PROGRAM PRG_09_PlcDiagnostic
VAR
	NetID						: 	STRING := '192.168.1.145.1.1';
	tonRecycle50ms				: 	TON;
	tonRecyclePublishMqtt		: 	TON;
	
	CpuMemoryUsage				:	ReadMemoryUsage;
	CpuUsageEx_Core2			:	TC_CPuUsageEx;
	CpuUsageEx_Core3			:	TC_CPuUsageEx;
	CpuLatencyEx_Core2			:	TC_SysLatencyEx;
	CpuLatencyEx_Core3			:	TC_SysLatencyEx;
	
	PlcDiagState				:	ARRAY [1..5] OF GenericState;
	
	{attribute 'OPC.UA.DA' := '0'}
	{attribute 'OPC.UA.DA.Access' := '1'}			// read only
	{attribute 'OPC.UA.DA.StructuredType' := '1'}
	PlcCpuMemUsageStruct		: SingleState_DataModel;
	
	{attribute 'OPC.UA.DA' := '0'}
	{attribute 'OPC.UA.DA.Access' := '1'}			// read only
	{attribute 'OPC.UA.DA.StructuredType' := '1'}
	PlcCpuCore2UsageStruct		: SingleState_DataModel;
	
	{attribute 'OPC.UA.DA' := '0'}
	{attribute 'OPC.UA.DA.Access' := '1'}			// read only
	{attribute 'OPC.UA.DA.StructuredType' := '1'}
	PlcCpuCore3UsageStruct		: SingleState_DataModel;
	
	{attribute 'OPC.UA.DA' := '0'}
	{attribute 'OPC.UA.DA.Access' := '1'}			// read only
	{attribute 'OPC.UA.DA.StructuredType' := '1'}
	PlcCpuCore2JitterStruct		: SingleState_DataModel;
	
	{attribute 'OPC.UA.DA' := '0'}
	{attribute 'OPC.UA.DA.Access' := '1'}			// read only
	{attribute 'OPC.UA.DA.StructuredType' := '1'}
	PlcCpuCore3JitterStruct		: SingleState_DataModel;

END_VAR


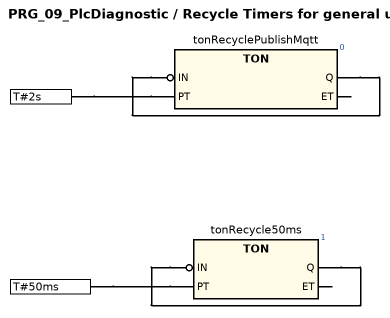
// PAGE Recycle Timers for general usage ---
tonRecyclePublishMqtt(IN := NOT tonRecyclePublishMqtt.Q, PT := T#2s); // TON
tonRecycle50ms(IN := NOT tonRecycle50ms.Q, PT := T#50ms); // TON

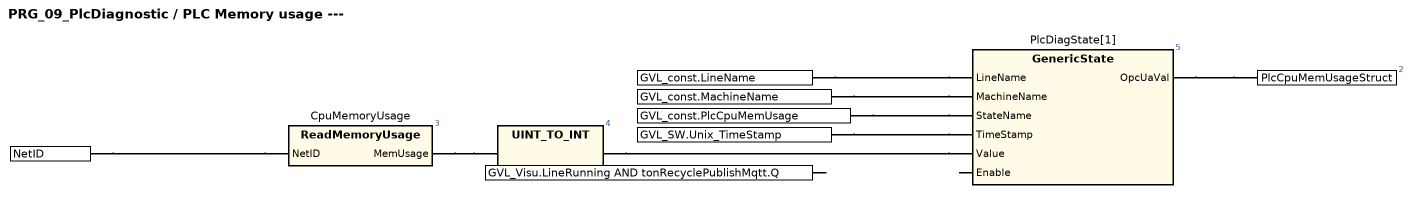
// PAGE PLC Memory usage ---
PlcCpuMemUsageStruct := PlcDiagState[1].OpcUaVal;
CpuMemoryUsage(NetID := NetID); // ReadMemoryUsage
PlcDiagState[1](
    LineName := GVL_const.LineName,
    MachineName := GVL_const.MachineName,
    StateName := GVL_const.PlcCpuMemUsage,
    TimeStamp := GVL_SW.Unix_TimeStamp,
    Value := UINT_TO_INT(CpuMemoryUsage.MemUsage)); // GenericState

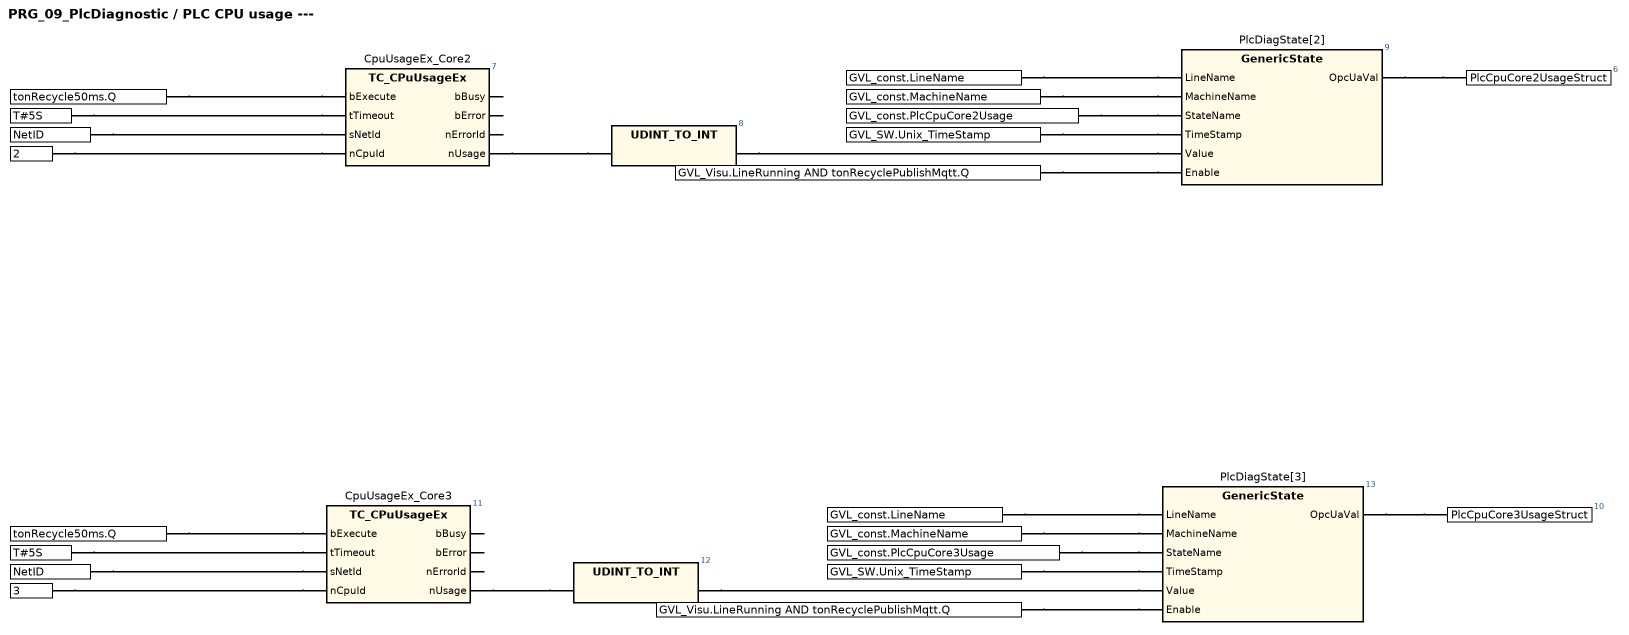
// PAGE PLC CPU usage ---
PlcCpuCore2UsageStruct := PlcDiagState[2].OpcUaVal;
CpuUsageEx_Core2(bExecute := tonRecycle50ms.Q, tTimeout := T#5S, sNetId := NetID, nCpuId := 2); // TC_CPuUsageEx
PlcDiagState[2](
    LineName := GVL_const.LineName,
    MachineName := GVL_const.MachineName,
    StateName := GVL_const.PlcCpuCore2Usage,
    TimeStamp := GVL_SW.Unix_TimeStamp,
    Value := UDINT_TO_INT(CpuUsageEx_Core2.nUsage),
    Enable := GVL_Visu.LineRunning AND tonRecyclePublishMqtt.Q); // GenericState
PlcCpuCore3UsageStruct := PlcDiagState[3].OpcUaVal;
CpuUsageEx_Core3(bExecute := tonRecycle50ms.Q, tTimeout := T#5S, sNetId := NetID, nCpuId := 3); // TC_CPuUsageEx
PlcDiagState[3](
    LineName := GVL_const.LineName,
    MachineName := GVL_const.MachineName,
    StateName := GVL_const.PlcCpuCore3Usage,
    TimeStamp := GVL_SW.Unix_TimeStamp,
    Value := UDINT_TO_INT(CpuUsageEx_Core3.nUsage),
    Enable := GVL_Visu.LineRunning AND tonRecyclePublishMqtt.Q); // GenericState

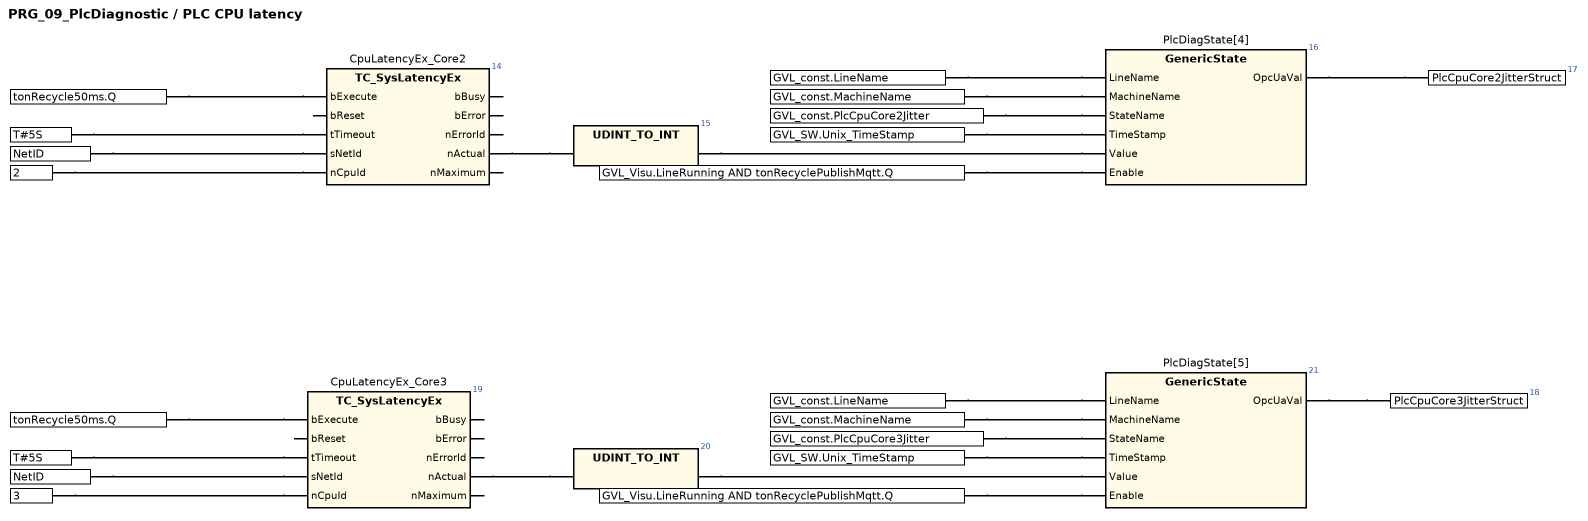
// PAGE PLC CPU latency
CpuLatencyEx_Core2(bExecute := tonRecycle50ms.Q, tTimeout := T#5S, sNetId := NetID, nCpuId := 2); // TC_SysLatencyEx
PlcDiagState[4](
    LineName := GVL_const.LineName,
    MachineName := GVL_const.MachineName,
    StateName := GVL_const.PlcCpuCore2Jitter,
    TimeStamp := GVL_SW.Unix_TimeStamp,
    Value := UDINT_TO_INT(CpuLatencyEx_Core2.nActual),
    Enable := GVL_Visu.LineRunning AND tonRecyclePublishMqtt.Q); // GenericState
PlcCpuCore2JitterStruct := PlcDiagState[4].OpcUaVal;
PlcCpuCore3JitterStruct := PlcDiagState[5].OpcUaVal;
CpuLatencyEx_Core3(bExecute := tonRecycle50ms.Q, tTimeout := T#5S, sNetId := NetID, nCpuId := 3); // TC_SysLatencyEx
PlcDiagState[5](
    LineName := GVL_const.LineName,
    MachineName := GVL_const.MachineName,
    StateName := GVL_const.PlcCpuCore3Jitter,
    TimeStamp := GVL_SW.Unix_TimeStamp,
    Value := UDINT_TO_INT(CpuLatencyEx_Core3.nActual),
    Enable := GVL_Visu.LineRunning AND tonRecyclePublishMqtt.Q); // GenericState
// GVL_Visu.LineRunning AND tonRecyclePublishMqtt.Q: input not connected

END_PROGRAM

(* stored: Version 1.1.0.1, ProductVersion 3.1.4024.15
   POU PRG_09_PlcDiagnostic: Id {52a30d09-a2c9-4a45-ab0a-0fa25ccb0a98}, SpecialFunc None *)
